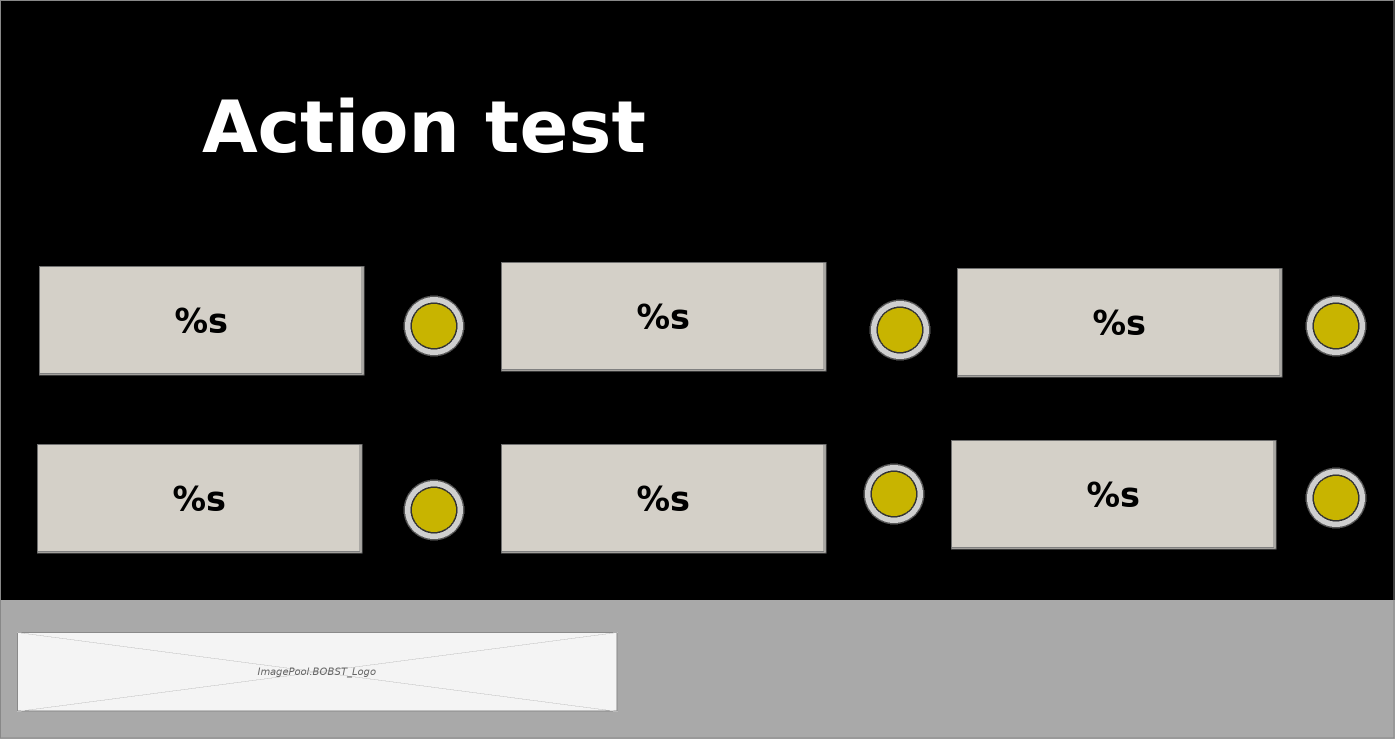
VISUALIZATION V_Test  // 1395x739
    Rectangle (-1,600 1396x140)
    Image (17,632 600x79), image: ImagePool.BOBST_Logo
        OnMouseDown: change screen: V_Menu
    Button (39,266 325x109), "%s", text variable: G_Visus.sTestFunction1
        OnMouseClick: execute { G_Visus.sTestBouton1 := True; }
    Button (501,262 325x109), "%s", text variable: G_Visus.sTestFunction2
        OnMouseClick: execute { G_Visus.sTestBouton2 := True; }
    Button (957,268 325x109), "%s", text variable: G_Visus.sTestFunction3
        OnMouseClick: execute { G_Visus.sTestBouton3 := True; }
    Button (37,444 325x109), "%s", text variable: G_Visus.sTestFunction4
        OnMouseClick: execute { G_Visus.sTestBouton4 := True; }
    Button (501,444 325x109), "%s", text variable: G_Visus.sTestFunction5
        OnMouseClick: execute { G_Visus.sTestBouton5 := True; }
    Button (951,440 325x109), "%s", text variable: G_Visus.sTestFunction6
        OnMouseClick: execute { G_Visus.sTestBouton6 := True; }
    Lamp1 (399,291 70x70), variable: G_Visus.sTestBouton1, style: Lamp-Lamp1-Yellow
    Lamp1 (865,295 70x70), variable: G_Visus.sTestBouton2, style: Lamp-Lamp1-Yellow
    Lamp1 (1301,291 70x70), variable: G_Visus.sTestBouton3, style: Lamp-Lamp1-Yellow
    Lamp1 (399,475 70x70), variable: G_Visus.sTestBouton4, style: Lamp-Lamp1-Yellow
    Lamp1 (859,459 70x70), variable: G_Visus.sTestBouton5, style: Lamp-Lamp1-Yellow
    Lamp1 (1301,463 70x70), variable: G_Visus.sTestBouton6, style: Lamp-Lamp1-Yellow
    Textfield (20,62 808x129), "Action test"
END_VISUALIZATION

(* stored: Version 1.1.0.1, ProductVersion 3.1.4024.12
   Visu V_Test: Id {2b32bbb8-d324-4d94-9429-e63ab8f1f3fa} *)
